// TIA Portal V17 export
// export: Created 2022-12-09T10:51:16.5558862Z, ExportSetting WithDefaults, DisplayName Totally Integrated Automation Portal, DisplayVersion V17 Update 5, DisplayName TIA Portal Openness, DisplayVersion V17 Update 5, DisplayName TIA Portal Version Control Interface, DisplayVersion V17, DisplayName Simotion SCOUT TIA, DisplayVersion 5.4.3.0, DisplayName SINAMICS Startdrive Advanced, DisplayVersion V17 SP1, DisplayName SINAMICS Startdrive G130, G150, S120, S150, SINAMICS MV, S210, DisplayVersion V17 SP1, DisplayName SINAMICS Startdrive G110M, G120, G120C, G120D, G120P, G115D, DisplayVersion V17 SP1, DisplayName STEP 7 Professional, DisplayVersion V17 Update 5, DisplayName STEP 7 Safety, DisplayVersion V17, DisplayName WinCC Advanced, DisplayVersion V17 Update 5
TYPE "NDSN_ST_Inventory"
// stored: IsFailsafeCompliant false
   STRUCT
      b_r_TempCtrl_Board1 : Bool;
      b_r_TempCtrl_Board2 : Bool;
      b_r_TempCtrl_Board3 : Bool;
      b_r_TempCtrl_Board4 : Bool;
      b_r_OEM_Unit : Bool;
      b_r_OLED_Unit : Bool;
      b_r_WIFI_Board : Bool;
      b_r_Refill_Board : Bool;
      b_r_Anybus_Board : Bool;
      b_r_Press_Sensor : Bool;
      b_r_Press_CtrlValve : Bool;
      i_r_NumOfTempZones_Internal : Int;
      i_r_NumOfTempZones_External : Int;
      i_r_NumOfMotors : Int;
      i_r_NumOfPumps : Int;
      i_r_NumOfATS : Int;
      i_r_NumOfWebClients : Int;
   END_STRUCT;
END_TYPE
